FUNCTION_BLOCK FB_Impulstest EXTENDS TcUnit.FB_TestSuite
VAR
	
END_VAR

//T01_TestDzialania ();

METHOD PRIVATE T01_TestDzialania
VAR_INST
	bUstawCzas: BOOL := TRUE;
	bWyjscie: BOOL;
	bKoniec: BOOL;
	rTimeOn		: REAL := 5000;
	rTimeOff	: REAL := 2500;
END_VAR
IF (TcUnit.TEST_ORDERED ('T01_TestDzialania')) THEN
	IF (bUstawCzas) THEN
		GVL.fbImpuls.SetTimeOn (rIN		:= rTimeOn);
		GVL.fbImpuls.SetTimeOff (rIN	:= rTimeOff);
		bUstawCzas						:= FALSE;
	END_IF
	GVL.fbImpuls ();
	
	bWyjscie							:= GVL.fbImpuls.GetExit ();
	
	IF (bKoniec) THEN
		TcUnit.TEST_FINISHED ();
	END_IF
END_IF
END_METHOD

END_FUNCTION_BLOCK

(* stored: Version 1.1.0.1, ProductVersion 3.1.4024.15
   POU FB_Impulstest: Id {cebafe51-2565-4de2-8e79-cb313cbe32b6}, SpecialFunc None
   Method T01_TestDzialania: Id {3f02e688-7f1b-41a7-8dd9-366eb05aabcd} *)
